KUKA KRL program: Mantenimiento.src, Mantenimiento.dat

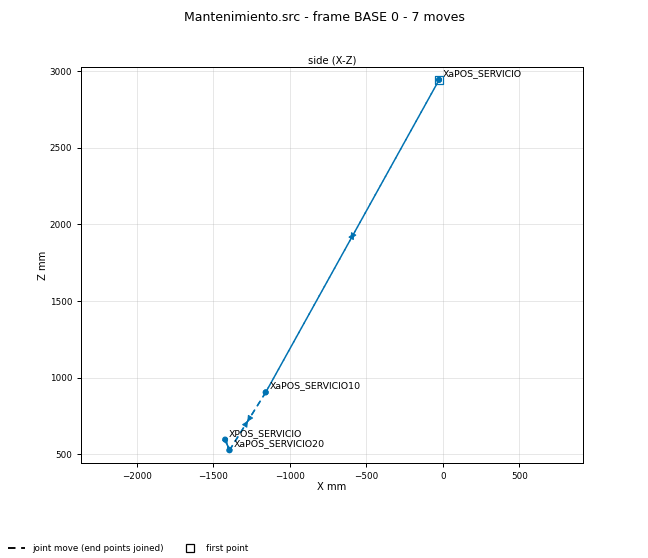
[picture p0: tool path of Mantenimiento.src in frame BASE 0, 7 of 9 moves have a stored position in this frame; points joined in program order, loops and branches not executed]
--- Mantenimiento.src ---
&ACCESS RVO1
&REL 25
&COMMENT PRG MANTENIMIENTO
&PARAM EDITMASK = *
&PARAM TEMPLATE = C:\KRC\Roboter\Template\vorgabe
&PARAM DISKPATH = KRC:\R1\Program\MAFELEC
DEF Mantenimiento( )
;FOLD INI;%{PE}
  ;FOLD BASISTECH INI
    GLOBAL INTERRUPT DECL 3 WHEN $STOPMESS==TRUE DO IR_STOPM ( )
    INTERRUPT ON 3
    BAS (#INITMOV,0 )
  ;ENDFOLD (BASISTECH INI)
;FOLD SPOTTECH INI
USERSPOT(#INIT)
;ENDFOLD (SPOTTECH INI)
;FOLD GRIPPERTECH INI
USER_GRP(0,DUMMY,DUMMY,GDEFAULT)
;ENDFOLD (GRIPPERTECH INI)
  ;FOLD USER INI
    ;Make your modifications here

  ;ENDFOLD (USER INI)
;ENDFOLD (INI)
;################################################
; PROYECTO: MAFELEC PLANTA DE BATERIAS
; ROBOT: 121_R1
; PROGRAMA: PROGRAMA DE SERVICIO
; CREADO POR: Alejandro Company(zaisor robotics)
; FECHA: 23-NOVIEMBRE-2022
; MODIFICADO POR:
; FECHA MODIFICACION: 13-ENERO-2023
;################################################

;FOLD PTP HOME Vel=100 % DEFAULT;%{PE}%R 8.3.48,%MKUKATPBASIS,%CMOVE,%VPTP,%P 1:PTP, 2:HOME, 3:, 5:100, 7:DEFAULT
$BWDSTART=FALSE
PDAT_ACT=PDEFAULT
FDAT_ACT=FHOME
BAS(#PTP_PARAMS,100)
$H_POS=XHOME
PTP XHOME
;ENDFOLD
Empujador(1,"R",FALSE)
Empujador(2,"R",FALSE)
Pines("R")

;FOLD PTP aPOS_SERVICIO Vel=20 % M Tool[9]:T_Gripper1_Vacio Base[0];%{PE}%R 8.3.48,%MKUKATPBASIS,%CMOVE,%VPTP,%P 1:PTP, 2:aPOS_SERVICIO, 3:, 5:20, 7:M
$BWDSTART=FALSE
PDAT_ACT=PM
FDAT_ACT=FaPOS_SERVICIO
BAS(#PTP_PARAMS,20)
PTP XaPOS_SERVICIO
;ENDFOLD
;FOLD PTP aPOS_SERVICIO10 CONT Vel=20 % M Tool[9]:T_Gripper1_Vacio Base[0];%{PE}%R 8.3.48,%MKUKATPBASIS,%CMOVE,%VPTP,%P 1:PTP, 2:aPOS_SERVICIO10, 3:C_DIS, 5:20, 7:M
$BWDSTART=FALSE
PDAT_ACT=PM
FDAT_ACT=FaPOS_SERVICIO10
BAS(#PTP_PARAMS,20)
PTP XaPOS_SERVICIO10 C_DIS
;ENDFOLD
;FOLD PTP aPOS_SERVICIO20 CONT Vel=20 % M Tool[9]:T_Gripper1_Vacio Base[0];%{PE}%R 8.3.48,%MKUKATPBASIS,%CMOVE,%VPTP,%P 1:PTP, 2:aPOS_SERVICIO20, 3:C_DIS, 5:20, 7:M
$BWDSTART=FALSE
PDAT_ACT=PM
FDAT_ACT=FaPOS_SERVICIO20
BAS(#PTP_PARAMS,20)
PTP XaPOS_SERVICIO20 C_DIS
;ENDFOLD

;POSICION DE SERVICIO
;FOLD PTP POS_SERVICIO Vel=20 % M Tool[9]:T_Gripper1_Vacio Base[0];%{PE}%R 8.3.48,%MKUKATPBASIS,%CMOVE,%VPTP,%P 1:PTP, 2:POS_SERVICIO, 3:, 5:20, 7:M
$BWDSTART=FALSE
PDAT_ACT=PM
FDAT_ACT=FPOS_SERVICIO
BAS(#PTP_PARAMS,20)
PTP XPOS_SERVICIO
;ENDFOLD
O_SERVP=TRUE


;ESPERA PERMISO RETORNO A HOME
WAIT FOR I_RETHP
O_SERVP=FALSE


;FOLD PTP aPOS_SERVICIO20 CONT Vel=20 % M Tool[9]:T_Gripper1_Vacio Base[0];%{PE}%R 8.3.48,%MKUKATPBASIS,%CMOVE,%VPTP,%P 1:PTP, 2:aPOS_SERVICIO20, 3:C_DIS, 5:20, 7:M
$BWDSTART=FALSE
PDAT_ACT=PM
FDAT_ACT=FaPOS_SERVICIO20
BAS(#PTP_PARAMS,20)
PTP XaPOS_SERVICIO20 C_DIS
;ENDFOLD
;FOLD PTP aPOS_SERVICIO10 CONT Vel=20 % M Tool[9]:T_Gripper1_Vacio Base[0];%{PE}%R 8.3.48,%MKUKATPBASIS,%CMOVE,%VPTP,%P 1:PTP, 2:aPOS_SERVICIO10, 3:C_DIS, 5:20, 7:M
$BWDSTART=FALSE
PDAT_ACT=PM
FDAT_ACT=FaPOS_SERVICIO10
BAS(#PTP_PARAMS,20)
PTP XaPOS_SERVICIO10 C_DIS
;ENDFOLD

;FOLD PTP aHOME Vel=20 % M Tool[9]:T_Gripper1_Vacio Base[0];%{PE}%R 8.3.48,%MKUKATPBASIS,%CMOVE,%VPTP,%P 1:PTP, 2:aHOME, 3:, 5:20, 7:M
$BWDSTART=FALSE
PDAT_ACT=PM
FDAT_ACT=FaHOME
BAS(#PTP_PARAMS,20)
PTP XaHOME
;ENDFOLD
;FOLD PTP HOME Vel=100 % DEFAULT;%{PE}%R 8.3.48,%MKUKATPBASIS,%CMOVE,%VPTP,%P 1:PTP, 2:HOME, 3:, 5:100, 7:DEFAULT
$BWDSTART=FALSE
PDAT_ACT=PDEFAULT
FDAT_ACT=FHOME
BAS(#PTP_PARAMS,100)
$H_POS=XHOME
PTP XHOME
;ENDFOLD
END

--- Mantenimiento.dat ---
&ACCESS RVO1
&REL 25
&COMMENT PRG MANTENIMIENTO
&PARAM EDITMASK = *
&PARAM TEMPLATE = C:\KRC\Roboter\Template\vorgabe
&PARAM DISKPATH = KRC:\R1\Program\MAFELEC
DEFDAT  Mantenimiento
;FOLD EXTERNAL DECLARATIONS;%{PE}%MKUKATPBASIS,%CEXT,%VCOMMON,%P
;FOLD GRIPPERTECH EXT
EXT  H50 (INT  :IN,INT  :IN,INT  :IN,GRP_TYP  :IN )
;ENDFOLD (GRIPPERTECH EXT)
;FOLD SPOTTECH EXT
EXT  USERSPOT (S_COMMAND  :IN,SPOT_TYPE  :IN )
;ENDFOLD (SPOTTECH EXT)
;FOLD BASISTECH EXT;%{PE}%MKUKATPBASIS,%CEXT,%VEXT,%P
EXT  BAS (BAS_COMMAND  :IN,REAL  :IN )
DECL INT SUCCESS
;ENDFOLD (BASISTECH EXT)
;FOLD USER EXT;%{E}%MKUKATPUSER,%CEXT,%VEXT,%P
;Make your modifications here

;ENDFOLD (USER EXT)
;ENDFOLD (EXTERNAL DECLARATIONS)
DECL BASIS_SUGG_T LAST_BASIS={POINT1[] "aPOS_SERVICIO10         ",POINT2[] "aPOS_SERVICIO10         ",CP_PARAMS[] "CPDAT0                  ",PTP_PARAMS[] "H                       ",CONT[] "C_DIS                   ",CP_VEL[] "2.0                     ",PTP_VEL[] "100                     ",SYNC_PARAMS[] "SYNCDAT                 ",SPL_NAME[] "S0                      ",A_PARAMS[] "ADAT0                   "}
DECL E6POS XPOS_SERVICIO={X -1423.22278,Y 12.1733541,Z 595.070862,A 13.3003607,B 1.31921577,C -179.688721,S 2,T 11,E1 0.0,E2 0.0,E3 0.0,E4 0.0,E5 0.0,E6 0.0}
DECL FDAT FPOS_SERVICIO={TOOL_NO 9,BASE_NO 0,IPO_FRAME #BASE,POINT2[] " ",TQ_STATE FALSE}
DECL PDAT PPDAT1={VEL 100.000,ACC 100.000,APO_DIST 100.000,GEAR_JERK 50.0000,EXAX_IGN 0}
DECL E6POS XAPOS_SERVICIO={X -25.0839577,Y -0.180477411,Z 2945.18604,A 176.393250,B 74.9027863,C -3.66209531,S 3,T 11,E1 0.0,E2 0.0,E3 0.0,E4 0.0,E5 0.0,E6 0.0}
DECL FDAT FaPOS_SERVICIO={TOOL_NO 9,BASE_NO 0,IPO_FRAME #BASE,POINT2[] " ",TQ_STATE FALSE}
DECL PDAT PH={VEL 100.000,ACC 100.000,APO_DIST 100.000,APO_MODE #CDIS,GEAR_JERK 50.0000,EXAX_IGN 0}
DECL E6POS XAHOME={X -25.0839252,Y -0.180477634,Z 2945.18604,A 176.393250,B 74.9027863,C -3.66209435,S 3,T 11,E1 0.0,E2 0.0,E3 0.0,E4 0.0,E5 0.0,E6 0.0}
DECL FDAT FaHOME={TOOL_NO 9,BASE_NO 0,IPO_FRAME #BASE,POINT2[] " ",TQ_STATE FALSE}
DECL PDAT PM={VEL 100.000,ACC 50.0000,APO_DIST 100.000,APO_MODE #CDIS,GEAR_JERK 50.0000,EXAX_IGN 0}
DECL E6POS XAPOS_SERVICIO10={X -1157.97717,Y -3.47961593,Z 903.077759,A 1.14985263,B -4.36971664,C 179.908035,S 2,T 11,E1 0.0,E2 0.0,E3 0.0,E4 0.0,E5 0.0,E6 0.0}
DECL FDAT FaPOS_SERVICIO10={TOOL_NO 9,BASE_NO 0,IPO_FRAME #BASE,POINT2[] " ",TQ_STATE FALSE}
DECL E6POS XAPOS_SERVICIO20={X -1394.66406,Y -3.47932601,Z 524.780518,A 1.14985144,B -4.36971664,C 179.908051,S 2,T 11,E1 0.0,E2 0.0,E3 0.0,E4 0.0,E5 0.0,E6 0.0}
DECL FDAT FaPOS_SERVICIO20={TOOL_NO 9,BASE_NO 0,IPO_FRAME #BASE,POINT2[] " ",TQ_STATE FALSE}
ENDDAT
